{attribute 'qualified_only'}
{attribute 'strict'}
TYPE eCapInsertStaState :
( 
	eUnknown := 51,
	eHoming,
	eDisabledReady,
	eWaitForVehicleTrigger,
	ePalletHoldDownGoingDown,
	ePalletHoldDownExtended,
	eCapSlideGoingDown,
	eCapSlideExtended,
	eCapSlideGoingUp,
	eCapSlideUp,
	ePalletHoldDownGoingUp,
	ePalletHoldDownUp,
	eDepart,
	eStopActive,
    eError
);
END_TYPE

(* stored: Version 1.1.0.1, ProductVersion 3.1.4022.6
   DUT eCapInsertStaState: Id {2f383e62-8410-4ffa-9477-3420ec5b6a6d} *)
